{attribute 'GeneratedUsingTerminal: EK1100-0000-0018'}
{attribute addProperty BoxType "EK1100-0000-0018"}
{attribute addProperty Id "Beckhoff_EL34xxEK1122Beckhoff_EL34xxEK1122_BFBD64DC2A_0001_EL3403_0000_0017EL3403_A37C91B877A_0002_EL3403_0000_0018EL3403_B537021B77A_0003_EL3403_0000_0019EL3403_B537021B77A_0004_EL3403_0000_0020EL3403_B537021B77A_0005_EL3403_0000_0021EL3403_B537021B77A_0006_EL3403_0000_0022EL3403_200C424073A_0007_EL3403_0000_0023EL3403_200C424073A_0008_EL3403_0010_0017EL3403_A37C91B877A_0009_EL3403_0010_0018EL3403_B537021B77A_0010_EL3403_0010_0019EL3403_B537021B77A_0011_EL3403_0010_0020EL3403_B537021B77A_0012_EL3403_0010_0021EL3403_B537021B77A_0013_EL3403_0010_0022EL3403_200C424073A_0014_EL3403_0010_0023EL3403_200C424073A_0015_EL3403_0010_0024EL3403_200C424073A_0016_EL3403_0026_0017EL3403_A37C91B877A_0017_EL3403_0026_0018EL3403_B537021B77A_0018_EL3403_0026_0019EL3403_B537021B77A_0019_EL3403_0026_0020EL3403_B537021B77A_0020_EL3403_0026_0021EL3403_B537021B77A_0021_EL3403_0026_0022EL3403_200C424073A_0022_EL3403_0026_0023EL3403_200C424073A_0023_EL3403_0026_0024EL3403_200C424073A_0024_EL3403_0100_0017EL3403_A37C91B877A_0025_EL3403_0100_0018EL3403_B537021B77A_0026_EL3403_0100_0019EL3403_B537021B77A_0027_EL3403_0100_0020EL3403_B537021B77A_0028_EL3403_0100_0021EL3403_B537021B77A_0029_EL3403_0100_0022EL3403_200C424073A_0030_EL3403_0100_0023EL3403_200C424073A_0031_EL3403_0100_0024EL3403_200C424073A_0032_EL3403_0111_0017EL3403_A37C91B877A_0033_EL3403_0111_0018EL3403_B537021B77A_0034_EL3403_0111_0019EL3403_B537021B77A_0035_EL3403_0111_0020EL3403_B537021B77A_0036_EL3403_0111_0021EL3403_B537021B77A_0037_EL3403_0111_0022EL3403_200C424073A_0038_EL3403_0111_0023EL3403_200C424073A_0039_EL3403_0111_0024EL3403_200C424073A_0040_EL3403_0126_0017EL3403_A37C91B877A_0041_EL3403_0126_0018EL3403_B537021B77A_0042_EL3403_0126_0019EL3403_B537021B77A_0043_EL3403_0126_0020EL3403_B537021B77A_0044_EL3403_0126_0021EL3403_B537021B77A_0045_EL3403_0126_0022EL3403_200C424073A_0046_EL3403_0126_0023EL3403_200C424073A_0047_EL3403_0126_0024EL3403_200C424073A_0048_EL3403_0333_0023EL3403_200C424073A_0049_EL3403_0333_0024EL3403_200C424073A_0050_EL3413_0000_0016EL3413_0563D89499A_0051_EL3413_0000_0017EL3413_0563D89499A_0052_EL3413_0000_0018EL3413_0563D89499A_0053_EL3413_0000_0019EL3413_0EB67A0F101A_0054_EL3413_0000_0020EL3413_0EB67A0F101A_0055_EL3413_0001_0016EL3413_0EB67A0F101A_0056_EL3413_0001_0017EL3413_0EB67A0F101A_0057_EL3413_0120_0017EL3413_0563D89499A_0058_EL3413_0001_0018EL3413_0EB67A0F101A_0059_EL3413_0120_0018EL3413_0EB67A0F101A_0060_EL3413_0120_0019EL3413_0EB67A0F101A_0061_EL3423_0000_0016EL3423_D53556D0190A_0062_EL3423_0000_0017EL3423_E7B0A427190A_0063_EL3423_0000_0018EL3423_E7B0A427190A_0064_EL3423_0000_0019EL3423_E7B0A427190A_0065_EL3423_0000_0020EL3423_8ADF1317118A_0066_EL3423_0000_0021EL3423_8ADF1317118A_0067_EL3433_0000_0016EL3433_0EB67A0F101A_0068_EL3433_0000_0017EL3433_0EB67A0F101A_0069_EL3433_0000_0018EL3433_0EB67A0F101A_0070_EL3443_0000_0016EL3443_696F77D6208A_0071_EL3443_0000_0017EL3443_721200EE208A_0072_EL3443_0000_0018EL3443_721200EE208A_0073_EL3443_0000_0019EL3443_721200EE208A_0074_EL3443_0000_0020EL3443_696F77D6208A_0075_EL3443_0000_0021EL3443_696F77D6208A_0076_EL3443_0010_0016EL3443_696F77D6208A_0077_EL3443_0010_0017EL3443_721200EE208A_0078_EL3443_0010_0018EL3443_721200EE208A_0079_EL3443_0010_0019EL3443_721200EE208A_0080_EL3443_0010_0020EL3443_696F77D6208A_0081_EL3443_0010_0021EL3443_696F77D6208A_0082_EL3443_0011_0018EL3443_721200EE208A_0083_EL3443_0011_0019EL3443_721200EE208A_0084_EL3443_0011_0020EL3443_696F77D6208A_0085_EL3443_0011_0021EL3443_696F77D6208A_0086_EL3443_0013_0018EL3443_721200EE208A_0087_EL3443_0013_0019EL3443_721200EE208A_0088_EL3443_0013_0020EL3443_696F77D6208A_0089_EL3443_0013_0021EL3443_696F77D6208A_0090_EL3446_0000_0016EL3446_D94D3CBC74A_0091_EL3446_0000_0017EL3446_D94D3CBC74A_0092_EL3453_0000_0017EL3453_C83104B4152A_0093_EL3453_0000_0018EL3453_24373016151A_0094_EL3453_0000_0019EL3453_24373016151A_0095_EL3453_0000_0020EL3453_C83104B4152A_0096_EL3453_0000_0021EL3453_C83104B4152A_0097_EL3453_0100_0021EL3453_C83104B4152A_0098_EL3483_0000_0016EL3483_E64A5C7841A_0099_EL3483_0000_0017EL3483_E64A5C7841A_0100_EL3483_0000_0018EL3483_E64A5C7841A_0101_EL3483_0000_0019EL3483_E64A5C7841A_0102_EL3483_0000_0020EL3483_E64A5C7841A_0103_EL3483_0000_0021EL3483_E64A5C7841A_0104_EL3483_0060_0018EL3483_2E666A7F65A_0105_EL3483_0060_0019EL3483_2E666A7F65A_0106_EL3483_0060_0020EL3483_A24D656565A_0107_EL3483_0060_0021EL3483_A24D656565"}
{attribute addProperty CRC "1552222167"}
{attribute addProperty Size "11825"}
TYPE Beckhoff_EL34xx_5C8507D7 EXTENDS EK1100_1FC0878B :
STRUCT
	{attribute addProperty Name "Beckhoff EL34xxEK1122"}
	{attribute addProperty PreviousPort "Beckhoff EL34xx : B"}
	Beckhoff_EL34xxEK1122 : Beckhoff_EL34xxEK1122_BFBD64DC;
	{attribute addProperty Name "A_0001(EL3403-0000-0017)"}
	{attribute addProperty PreviousPort "Beckhoff EL34xxEK1122 : C"}
	A_0001_EL3403_0000_0017 : EL3403_A37C91B8;
	{attribute addProperty Name "A_0002(EL3403-0000-0018)"}
	{attribute addProperty PreviousPort "A_0001(EL3403-0000-0017) : B"}
	A_0002_EL3403_0000_0018 : EL3403_B537021B;
	{attribute addProperty Name "A_0003(EL3403-0000-0019)"}
	{attribute addProperty PreviousPort "A_0002(EL3403-0000-0018) : B"}
	A_0003_EL3403_0000_0019 : EL3403_B537021B;
	{attribute addProperty Name "A_0004(EL3403-0000-0020)"}
	{attribute addProperty PreviousPort "A_0003(EL3403-0000-0019) : B"}
	A_0004_EL3403_0000_0020 : EL3403_B537021B;
	{attribute addProperty Name "A_0005(EL3403-0000-0021)"}
	{attribute addProperty PreviousPort "A_0004(EL3403-0000-0020) : B"}
	A_0005_EL3403_0000_0021 : EL3403_B537021B;
	{attribute addProperty Name "A_0006(EL3403-0000-0022)"}
	{attribute addProperty PreviousPort "A_0005(EL3403-0000-0021) : B"}
	A_0006_EL3403_0000_0022 : EL3403_200C4240;
	{attribute addProperty Name "A_0007(EL3403-0000-0023)"}
	{attribute addProperty PreviousPort "A_0006(EL3403-0000-0022) : B"}
	A_0007_EL3403_0000_0023 : EL3403_200C4240;
	{attribute addProperty Name "A_0008(EL3403-0010-0017)"}
	{attribute addProperty PreviousPort "A_0007(EL3403-0000-0023) : B"}
	A_0008_EL3403_0010_0017 : EL3403_A37C91B8;
	{attribute addProperty Name "A_0009(EL3403-0010-0018)"}
	{attribute addProperty PreviousPort "A_0008(EL3403-0010-0017) : B"}
	A_0009_EL3403_0010_0018 : EL3403_B537021B;
	{attribute addProperty Name "A_0010(EL3403-0010-0019)"}
	{attribute addProperty PreviousPort "A_0009(EL3403-0010-0018) : B"}
	A_0010_EL3403_0010_0019 : EL3403_B537021B;
	{attribute addProperty Name "A_0011(EL3403-0010-0020)"}
	{attribute addProperty PreviousPort "A_0010(EL3403-0010-0019) : B"}
	A_0011_EL3403_0010_0020 : EL3403_B537021B;
	{attribute addProperty Name "A_0012(EL3403-0010-0021)"}
	{attribute addProperty PreviousPort "A_0011(EL3403-0010-0020) : B"}
	A_0012_EL3403_0010_0021 : EL3403_B537021B;
	{attribute addProperty Name "A_0013(EL3403-0010-0022)"}
	{attribute addProperty PreviousPort "A_0012(EL3403-0010-0021) : B"}
	A_0013_EL3403_0010_0022 : EL3403_200C4240;
	{attribute addProperty Name "A_0014(EL3403-0010-0023)"}
	{attribute addProperty PreviousPort "A_0013(EL3403-0010-0022) : B"}
	A_0014_EL3403_0010_0023 : EL3403_200C4240;
	{attribute addProperty Name "A_0015(EL3403-0010-0024)"}
	{attribute addProperty PreviousPort "A_0014(EL3403-0010-0023) : B"}
	A_0015_EL3403_0010_0024 : EL3403_200C4240;
	{attribute addProperty Name "A_0016(EL3403-0026-0017)"}
	{attribute addProperty PreviousPort "A_0015(EL3403-0010-0024) : B"}
	A_0016_EL3403_0026_0017 : EL3403_A37C91B8;
	{attribute addProperty Name "A_0017(EL3403-0026-0018)"}
	{attribute addProperty PreviousPort "A_0016(EL3403-0026-0017) : B"}
	A_0017_EL3403_0026_0018 : EL3403_B537021B;
	{attribute addProperty Name "A_0018(EL3403-0026-0019)"}
	{attribute addProperty PreviousPort "A_0017(EL3403-0026-0018) : B"}
	A_0018_EL3403_0026_0019 : EL3403_B537021B;
	{attribute addProperty Name "A_0019(EL3403-0026-0020)"}
	{attribute addProperty PreviousPort "A_0018(EL3403-0026-0019) : B"}
	A_0019_EL3403_0026_0020 : EL3403_B537021B;
	{attribute addProperty Name "A_0020(EL3403-0026-0021)"}
	{attribute addProperty PreviousPort "A_0019(EL3403-0026-0020) : B"}
	A_0020_EL3403_0026_0021 : EL3403_B537021B;
	{attribute addProperty Name "A_0021(EL3403-0026-0022)"}
	{attribute addProperty PreviousPort "A_0020(EL3403-0026-0021) : B"}
	A_0021_EL3403_0026_0022 : EL3403_200C4240;
	{attribute addProperty Name "A_0022(EL3403-0026-0023)"}
	{attribute addProperty PreviousPort "A_0021(EL3403-0026-0022) : B"}
	A_0022_EL3403_0026_0023 : EL3403_200C4240;
	{attribute addProperty Name "A_0023(EL3403-0026-0024)"}
	{attribute addProperty PreviousPort "A_0022(EL3403-0026-0023) : B"}
	A_0023_EL3403_0026_0024 : EL3403_200C4240;
	{attribute addProperty Name "A_0024(EL3403-0100-0017)"}
	{attribute addProperty PreviousPort "A_0023(EL3403-0026-0024) : B"}
	A_0024_EL3403_0100_0017 : EL3403_A37C91B8;
	{attribute addProperty Name "A_0025(EL3403-0100-0018)"}
	{attribute addProperty PreviousPort "A_0024(EL3403-0100-0017) : B"}
	A_0025_EL3403_0100_0018 : EL3403_B537021B;
	{attribute addProperty Name "A_0026(EL3403-0100-0019)"}
	{attribute addProperty PreviousPort "A_0025(EL3403-0100-0018) : B"}
	A_0026_EL3403_0100_0019 : EL3403_B537021B;
	{attribute addProperty Name "A_0027(EL3403-0100-0020)"}
	{attribute addProperty PreviousPort "A_0026(EL3403-0100-0019) : B"}
	A_0027_EL3403_0100_0020 : EL3403_B537021B;
	{attribute addProperty Name "A_0028(EL3403-0100-0021)"}
	{attribute addProperty PreviousPort "A_0027(EL3403-0100-0020) : B"}
	A_0028_EL3403_0100_0021 : EL3403_B537021B;
	{attribute addProperty Name "A_0029(EL3403-0100-0022)"}
	{attribute addProperty PreviousPort "A_0028(EL3403-0100-0021) : B"}
	A_0029_EL3403_0100_0022 : EL3403_200C4240;
	{attribute addProperty Name "A_0030(EL3403-0100-0023)"}
	{attribute addProperty PreviousPort "A_0029(EL3403-0100-0022) : B"}
	A_0030_EL3403_0100_0023 : EL3403_200C4240;
	{attribute addProperty Name "A_0031(EL3403-0100-0024)"}
	{attribute addProperty PreviousPort "A_0030(EL3403-0100-0023) : B"}
	A_0031_EL3403_0100_0024 : EL3403_200C4240;
	{attribute addProperty Name "A_0032(EL3403-0111-0017)"}
	{attribute addProperty PreviousPort "A_0031(EL3403-0100-0024) : B"}
	A_0032_EL3403_0111_0017 : EL3403_A37C91B8;
	{attribute addProperty Name "A_0033(EL3403-0111-0018)"}
	{attribute addProperty PreviousPort "A_0032(EL3403-0111-0017) : B"}
	A_0033_EL3403_0111_0018 : EL3403_B537021B;
	{attribute addProperty Name "A_0034(EL3403-0111-0019)"}
	{attribute addProperty PreviousPort "A_0033(EL3403-0111-0018) : B"}
	A_0034_EL3403_0111_0019 : EL3403_B537021B;
	{attribute addProperty Name "A_0035(EL3403-0111-0020)"}
	{attribute addProperty PreviousPort "A_0034(EL3403-0111-0019) : B"}
	A_0035_EL3403_0111_0020 : EL3403_B537021B;
	{attribute addProperty Name "A_0036(EL3403-0111-0021)"}
	{attribute addProperty PreviousPort "A_0035(EL3403-0111-0020) : B"}
	A_0036_EL3403_0111_0021 : EL3403_B537021B;
	{attribute addProperty Name "A_0037(EL3403-0111-0022)"}
	{attribute addProperty PreviousPort "A_0036(EL3403-0111-0021) : B"}
	A_0037_EL3403_0111_0022 : EL3403_200C4240;
	{attribute addProperty Name "A_0038(EL3403-0111-0023)"}
	{attribute addProperty PreviousPort "A_0037(EL3403-0111-0022) : B"}
	A_0038_EL3403_0111_0023 : EL3403_200C4240;
	{attribute addProperty Name "A_0039(EL3403-0111-0024)"}
	{attribute addProperty PreviousPort "A_0038(EL3403-0111-0023) : B"}
	A_0039_EL3403_0111_0024 : EL3403_200C4240;
	{attribute addProperty Name "A_0040(EL3403-0126-0017)"}
	{attribute addProperty PreviousPort "A_0039(EL3403-0111-0024) : B"}
	A_0040_EL3403_0126_0017 : EL3403_A37C91B8;
	{attribute addProperty Name "A_0041(EL3403-0126-0018)"}
	{attribute addProperty PreviousPort "A_0040(EL3403-0126-0017) : B"}
	A_0041_EL3403_0126_0018 : EL3403_B537021B;
	{attribute addProperty Name "A_0042(EL3403-0126-0019)"}
	{attribute addProperty PreviousPort "A_0041(EL3403-0126-0018) : B"}
	A_0042_EL3403_0126_0019 : EL3403_B537021B;
	{attribute addProperty Name "A_0043(EL3403-0126-0020)"}
	{attribute addProperty PreviousPort "A_0042(EL3403-0126-0019) : B"}
	A_0043_EL3403_0126_0020 : EL3403_B537021B;
	{attribute addProperty Name "A_0044(EL3403-0126-0021)"}
	{attribute addProperty PreviousPort "A_0043(EL3403-0126-0020) : B"}
	A_0044_EL3403_0126_0021 : EL3403_B537021B;
	{attribute addProperty Name "A_0045(EL3403-0126-0022)"}
	{attribute addProperty PreviousPort "A_0044(EL3403-0126-0021) : B"}
	A_0045_EL3403_0126_0022 : EL3403_200C4240;
	{attribute addProperty Name "A_0046(EL3403-0126-0023)"}
	{attribute addProperty PreviousPort "A_0045(EL3403-0126-0022) : B"}
	A_0046_EL3403_0126_0023 : EL3403_200C4240;
	{attribute addProperty Name "A_0047(EL3403-0126-0024)"}
	{attribute addProperty PreviousPort "A_0046(EL3403-0126-0023) : B"}
	A_0047_EL3403_0126_0024 : EL3403_200C4240;
	{attribute addProperty Name "A_0048(EL3403-0333-0023)"}
	{attribute addProperty PreviousPort "A_0047(EL3403-0126-0024) : B"}
	A_0048_EL3403_0333_0023 : EL3403_200C4240;
	{attribute addProperty Name "A_0049(EL3403-0333-0024)"}
	{attribute addProperty PreviousPort "A_0048(EL3403-0333-0023) : B"}
	A_0049_EL3403_0333_0024 : EL3403_200C4240;
	{attribute addProperty Name "A_0050(EL3413-0000-0016)"}
	{attribute addProperty PreviousPort "A_0049(EL3403-0333-0024) : B"}
	A_0050_EL3413_0000_0016 : EL3413_0563D894;
	{attribute addProperty Name "A_0051(EL3413-0000-0017)"}
	{attribute addProperty PreviousPort "A_0050(EL3413-0000-0016) : B"}
	A_0051_EL3413_0000_0017 : EL3413_0563D894;
	{attribute addProperty Name "A_0052(EL3413-0000-0018)"}
	{attribute addProperty PreviousPort "A_0051(EL3413-0000-0017) : B"}
	A_0052_EL3413_0000_0018 : EL3413_0563D894;
	{attribute addProperty Name "A_0053(EL3413-0000-0019)"}
	{attribute addProperty PreviousPort "A_0052(EL3413-0000-0018) : B"}
	A_0053_EL3413_0000_0019 : EL3413_0EB67A0F;
	{attribute addProperty Name "A_0054(EL3413-0000-0020)"}
	{attribute addProperty PreviousPort "A_0053(EL3413-0000-0019) : B"}
	A_0054_EL3413_0000_0020 : EL3413_0EB67A0F;
	{attribute addProperty Name "A_0055(EL3413-0001-0016)"}
	{attribute addProperty PreviousPort "A_0054(EL3413-0000-0020) : B"}
	A_0055_EL3413_0001_0016 : EL3413_0EB67A0F;
	{attribute addProperty Name "A_0056(EL3413-0001-0017)"}
	{attribute addProperty PreviousPort "A_0055(EL3413-0001-0016) : B"}
	A_0056_EL3413_0001_0017 : EL3413_0EB67A0F;
	{attribute addProperty Name "A_0057(EL3413-0120-0017)"}
	{attribute addProperty PreviousPort "A_0056(EL3413-0001-0017) : B"}
	A_0057_EL3413_0120_0017 : EL3413_0563D894;
	{attribute addProperty Name "A_0058(EL3413-0001-0018)"}
	{attribute addProperty PreviousPort "A_0057(EL3413-0120-0017) : B"}
	A_0058_EL3413_0001_0018 : EL3413_0EB67A0F;
	{attribute addProperty Name "A_0059(EL3413-0120-0018)"}
	{attribute addProperty PreviousPort "A_0058(EL3413-0001-0018) : B"}
	A_0059_EL3413_0120_0018 : EL3413_0EB67A0F;
	{attribute addProperty Name "A_0060(EL3413-0120-0019)"}
	{attribute addProperty PreviousPort "A_0059(EL3413-0120-0018) : B"}
	A_0060_EL3413_0120_0019 : EL3413_0EB67A0F;
	{attribute addProperty Name "A_0061(EL3423-0000-0016)"}
	{attribute addProperty PreviousPort "A_0060(EL3413-0120-0019) : B"}
	A_0061_EL3423_0000_0016 : EL3423_D53556D0;
	{attribute addProperty Name "A_0062(EL3423-0000-0017)"}
	{attribute addProperty PreviousPort "A_0061(EL3423-0000-0016) : B"}
	A_0062_EL3423_0000_0017 : EL3423_E7B0A427;
	{attribute addProperty Name "A_0063(EL3423-0000-0018)"}
	{attribute addProperty PreviousPort "A_0062(EL3423-0000-0017) : B"}
	A_0063_EL3423_0000_0018 : EL3423_E7B0A427;
	{attribute addProperty Name "A_0064(EL3423-0000-0019)"}
	{attribute addProperty PreviousPort "A_0063(EL3423-0000-0018) : B"}
	A_0064_EL3423_0000_0019 : EL3423_E7B0A427;
	{attribute addProperty Name "A_0065(EL3423-0000-0020)"}
	{attribute addProperty PreviousPort "A_0064(EL3423-0000-0019) : B"}
	A_0065_EL3423_0000_0020 : EL3423_8ADF1317;
	{attribute addProperty Name "A_0066(EL3423-0000-0021)"}
	{attribute addProperty PreviousPort "A_0065(EL3423-0000-0020) : B"}
	A_0066_EL3423_0000_0021 : EL3423_8ADF1317;
	{attribute addProperty Name "A_0067(EL3433-0000-0016)"}
	{attribute addProperty PreviousPort "A_0066(EL3423-0000-0021) : B"}
	A_0067_EL3433_0000_0016 : EL3433_0EB67A0F;
	{attribute addProperty Name "A_0068(EL3433-0000-0017)"}
	{attribute addProperty PreviousPort "A_0067(EL3433-0000-0016) : B"}
	A_0068_EL3433_0000_0017 : EL3433_0EB67A0F;
	{attribute addProperty Name "A_0069(EL3433-0000-0018)"}
	{attribute addProperty PreviousPort "A_0068(EL3433-0000-0017) : B"}
	A_0069_EL3433_0000_0018 : EL3433_0EB67A0F;
	{attribute addProperty Name "A_0070(EL3443-0000-0016)"}
	{attribute addProperty PreviousPort "A_0069(EL3433-0000-0018) : B"}
	A_0070_EL3443_0000_0016 : EL3443_696F77D6;
	{attribute addProperty Name "A_0071(EL3443-0000-0017)"}
	{attribute addProperty PreviousPort "A_0070(EL3443-0000-0016) : B"}
	A_0071_EL3443_0000_0017 : EL3443_721200EE;
	{attribute addProperty Name "A_0072(EL3443-0000-0018)"}
	{attribute addProperty PreviousPort "A_0071(EL3443-0000-0017) : B"}
	A_0072_EL3443_0000_0018 : EL3443_721200EE;
	{attribute addProperty Name "A_0073(EL3443-0000-0019)"}
	{attribute addProperty PreviousPort "A_0072(EL3443-0000-0018) : B"}
	A_0073_EL3443_0000_0019 : EL3443_721200EE;
	{attribute addProperty Name "A_0074(EL3443-0000-0020)"}
	{attribute addProperty PreviousPort "A_0073(EL3443-0000-0019) : B"}
	A_0074_EL3443_0000_0020 : EL3443_696F77D6;
	{attribute addProperty Name "A_0075(EL3443-0000-0021)"}
	{attribute addProperty PreviousPort "A_0074(EL3443-0000-0020) : B"}
	A_0075_EL3443_0000_0021 : EL3443_696F77D6;
	{attribute addProperty Name "A_0076(EL3443-0010-0016)"}
	{attribute addProperty PreviousPort "A_0075(EL3443-0000-0021) : B"}
	A_0076_EL3443_0010_0016 : EL3443_696F77D6;
	{attribute addProperty Name "A_0077(EL3443-0010-0017)"}
	{attribute addProperty PreviousPort "A_0076(EL3443-0010-0016) : B"}
	A_0077_EL3443_0010_0017 : EL3443_721200EE;
	{attribute addProperty Name "A_0078(EL3443-0010-0018)"}
	{attribute addProperty PreviousPort "A_0077(EL3443-0010-0017) : B"}
	A_0078_EL3443_0010_0018 : EL3443_721200EE;
	{attribute addProperty Name "A_0079(EL3443-0010-0019)"}
	{attribute addProperty PreviousPort "A_0078(EL3443-0010-0018) : B"}
	A_0079_EL3443_0010_0019 : EL3443_721200EE;
	{attribute addProperty Name "A_0080(EL3443-0010-0020)"}
	{attribute addProperty PreviousPort "A_0079(EL3443-0010-0019) : B"}
	A_0080_EL3443_0010_0020 : EL3443_696F77D6;
	{attribute addProperty Name "A_0081(EL3443-0010-0021)"}
	{attribute addProperty PreviousPort "A_0080(EL3443-0010-0020) : B"}
	A_0081_EL3443_0010_0021 : EL3443_696F77D6;
	{attribute addProperty Name "A_0082(EL3443-0011-0018)"}
	{attribute addProperty PreviousPort "A_0081(EL3443-0010-0021) : B"}
	A_0082_EL3443_0011_0018 : EL3443_721200EE;
	{attribute addProperty Name "A_0083(EL3443-0011-0019)"}
	{attribute addProperty PreviousPort "A_0082(EL3443-0011-0018) : B"}
	A_0083_EL3443_0011_0019 : EL3443_721200EE;
	{attribute addProperty Name "A_0084(EL3443-0011-0020)"}
	{attribute addProperty PreviousPort "A_0083(EL3443-0011-0019) : B"}
	A_0084_EL3443_0011_0020 : EL3443_696F77D6;
	{attribute addProperty Name "A_0085(EL3443-0011-0021)"}
	{attribute addProperty PreviousPort "A_0084(EL3443-0011-0020) : B"}
	A_0085_EL3443_0011_0021 : EL3443_696F77D6;
	{attribute addProperty Name "A_0086(EL3443-0013-0018)"}
	{attribute addProperty PreviousPort "A_0085(EL3443-0011-0021) : B"}
	A_0086_EL3443_0013_0018 : EL3443_721200EE;
	{attribute addProperty Name "A_0087(EL3443-0013-0019)"}
	{attribute addProperty PreviousPort "A_0086(EL3443-0013-0018) : B"}
	A_0087_EL3443_0013_0019 : EL3443_721200EE;
	{attribute addProperty Name "A_0088(EL3443-0013-0020)"}
	{attribute addProperty PreviousPort "A_0087(EL3443-0013-0019) : B"}
	A_0088_EL3443_0013_0020 : EL3443_696F77D6;
	{attribute addProperty Name "A_0089(EL3443-0013-0021)"}
	{attribute addProperty PreviousPort "A_0088(EL3443-0013-0020) : B"}
	A_0089_EL3443_0013_0021 : EL3443_696F77D6;
	{attribute addProperty Name "A_0090(EL3446-0000-0016)"}
	{attribute addProperty PreviousPort "A_0089(EL3443-0013-0021) : B"}
	A_0090_EL3446_0000_0016 : EL3446_D94D3CBC;
	{attribute addProperty Name "A_0091(EL3446-0000-0017)"}
	{attribute addProperty PreviousPort "A_0090(EL3446-0000-0016) : B"}
	A_0091_EL3446_0000_0017 : EL3446_D94D3CBC;
	{attribute addProperty Name "A_0092(EL3453-0000-0017)"}
	{attribute addProperty PreviousPort "A_0091(EL3446-0000-0017) : B"}
	A_0092_EL3453_0000_0017 : EL3453_C83104B4;
	{attribute addProperty Name "A_0093(EL3453-0000-0018)"}
	{attribute addProperty PreviousPort "A_0092(EL3453-0000-0017) : B"}
	A_0093_EL3453_0000_0018 : EL3453_24373016;
	{attribute addProperty Name "A_0094(EL3453-0000-0019)"}
	{attribute addProperty PreviousPort "A_0093(EL3453-0000-0018) : B"}
	A_0094_EL3453_0000_0019 : EL3453_24373016;
	{attribute addProperty Name "A_0095(EL3453-0000-0020)"}
	{attribute addProperty PreviousPort "A_0094(EL3453-0000-0019) : B"}
	A_0095_EL3453_0000_0020 : EL3453_C83104B4;
	{attribute addProperty Name "A_0096(EL3453-0000-0021)"}
	{attribute addProperty PreviousPort "A_0095(EL3453-0000-0020) : B"}
	A_0096_EL3453_0000_0021 : EL3453_C83104B4;
	{attribute addProperty Name "A_0097(EL3453-0100-0021)"}
	{attribute addProperty PreviousPort "A_0096(EL3453-0000-0021) : B"}
	A_0097_EL3453_0100_0021 : EL3453_C83104B4;
	{attribute addProperty Name "A_0098(EL3483-0000-0016)"}
	{attribute addProperty PreviousPort "A_0097(EL3453-0100-0021) : B"}
	A_0098_EL3483_0000_0016 : EL3483_E64A5C78;
	{attribute addProperty Name "A_0099(EL3483-0000-0017)"}
	{attribute addProperty PreviousPort "A_0098(EL3483-0000-0016) : B"}
	A_0099_EL3483_0000_0017 : EL3483_E64A5C78;
	{attribute addProperty Name "A_0100(EL3483-0000-0018)"}
	{attribute addProperty PreviousPort "A_0099(EL3483-0000-0017) : B"}
	A_0100_EL3483_0000_0018 : EL3483_E64A5C78;
	{attribute addProperty Name "A_0101(EL3483-0000-0019)"}
	{attribute addProperty PreviousPort "A_0100(EL3483-0000-0018) : B"}
	A_0101_EL3483_0000_0019 : EL3483_E64A5C78;
	{attribute addProperty Name "A_0102(EL3483-0000-0020)"}
	{attribute addProperty PreviousPort "A_0101(EL3483-0000-0019) : B"}
	A_0102_EL3483_0000_0020 : EL3483_E64A5C78;
	{attribute addProperty Name "A_0103(EL3483-0000-0021)"}
	{attribute addProperty PreviousPort "A_0102(EL3483-0000-0020) : B"}
	A_0103_EL3483_0000_0021 : EL3483_E64A5C78;
	{attribute addProperty Name "A_0104(EL3483-0060-0018)"}
	{attribute addProperty PreviousPort "A_0103(EL3483-0000-0021) : B"}
	A_0104_EL3483_0060_0018 : EL3483_2E666A7F;
	{attribute addProperty Name "A_0105(EL3483-0060-0019)"}
	{attribute addProperty PreviousPort "A_0104(EL3483-0060-0018) : B"}
	A_0105_EL3483_0060_0019 : EL3483_2E666A7F;
	{attribute addProperty Name "A_0106(EL3483-0060-0020)"}
	{attribute addProperty PreviousPort "A_0105(EL3483-0060-0019) : B"}
	A_0106_EL3483_0060_0020 : EL3483_A24D6565;
	{attribute addProperty Name "A_0107(EL3483-0060-0021)"}
	{attribute addProperty PreviousPort "A_0106(EL3483-0060-0020) : B"}
	A_0107_EL3483_0060_0021 : EL3483_A24D6565;
END_STRUCT
END_TYPE

(* stored: Version 1.2.0.0, ProductVersion 3.1.4024.11
   DUT Beckhoff_EL34xx_5C8507D7: Id {4d51acaf-3082-42df-9c09-001c6357e835} *)
